FUNCTION_BLOCK CycleCount
VAR
	Picked : BOOL;
	
END_VAR

METHOD mPicked : BOOL
VAR_INPUT
END_VAR
Picked := TRUE;
END_METHOD

PROPERTY pPicked : BOOL
GET
pPicked := Picked;
END_GET
SET
Picked := pPicked;
END_SET
END_PROPERTY

END_FUNCTION_BLOCK

(* stored: Version 1.1.0.1, ProductVersion 3.1.4024.9
   POU CycleCount: Id {039ed861-983f-49d3-8a50-019c0e5337db}, SpecialFunc None
   Method mPicked: Id {6a453c49-015c-4cfc-b486-4d21afa9f438}
   Property pPicked: Id {53b276ee-24ff-44ce-a4c3-a4058d5e5935}
   Get Get: Id {5e01d6f1-6fc8-4bee-be2d-d684e0bc32e1}
   Set Set: Id {f9ac3772-6d28-497f-a44a-e60f68cb282f} *)
